TYPE ST_MethodOut :  //    方法
STRUCT
             Execute            :BOOL;  
             Done1               :BOOL;  
             Done2               :BOOL;  
             Error               :BOOL;

END_STRUCT
END_TYPE

(* stored: Version 1.1.0.1, ProductVersion 3.1.4024.9
   DUT ST_MethodOut: Id {327e3b12-400f-4ddd-bdf6-a1f16727ed7b} *)
